VAR_GLOBAL
    (* OverrideMode *)
    {attribute 'pytmc' := 'pv: UED:RCC:VAC:OVRD_MODE'}
    xSystemOverrideMode_RCC	: BOOL := FALSE;

    (* Roughing Manifold Valvese *)

    {attribute 'pytmc' :=' pv: UED:RCC:VRC:01 '}
    {attribute 'TcLinkTo' := 	'.i_xClsLS	:=  TIID^Device 1 (EtherCAT)^Term 1 (EK1200)^RCC_E2 (EL1004)^Channel 1^Input;
                                .q_xOPN_DO	:=	TIID^Device 1 (EtherCAT)^Term 1 (EK1200)^RCC_E1 (EL2004)^Channel 1^Output'}
    RCC_VRC_01 : FB_VRC_NC_ClsLS;

    (* Roughing Manifold Valvese *)

    {attribute 'pytmc' :=' pv: UED:RCC:VRC:02 '}
    {attribute 'TcLinkTo' := 	'.i_xOpnLS	:= 	TIID^Device 1 (EtherCAT)^Term 1 (EK1200)^RCC_E2 (EL1004)^Channel 3^Input;
                                 .i_xClsLS	:=	TIID^Device 1 (EtherCAT)^Term 1 (EK1200)^RCC_E2 (EL1004)^Channel 4^Input;
                                .q_xOPN_DO	:=	TIID^Device 1 (EtherCAT)^Term 1 (EK1200)^RCC_E1 (EL2004)^Channel 2^Output'}
    RCC_VRC_02 : FB_VRC;

    (* Roughing Manifold Valvese *)

    {attribute 'pytmc' :=' pv: UED:RCC:VRC:03 '}
    {attribute 'TcLinkTo' := 	'.i_xClsLS	:=	TIID^Device 1 (EtherCAT)^Term 1 (EK1200)^RCC_E3 (EL1004)^Channel 1^Input;
                                .q_xOPN_DO	:= 	TIID^Device 1 (EtherCAT)^Term 1 (EK1200)^RCC_E1 (EL2004)^Channel 3^Output'}
    RCC_VRC_03 : FB_VRC_NC_ClsLS;

    (* Roughing Manifold Valvese *)

    {attribute 'pytmc' :=' pv: UED:RCC:VRC:04 '}
    {attribute 'TcLinkTo' := 	'.i_xClsLS	:=	TIID^Device 1 (EtherCAT)^Term 1 (EK1200)^RCC_E3 (EL1004)^Channel 1^Input;
                                .q_xOPN_DO	:=  TIID^Device 1 (EtherCAT)^Term 1 (EK1200)^RCC_E1 (EL2004)^Channel 4^Output'}
    RCC_VRC_04 : FB_VRC_NC_ClsLS;


    {attribute 'pytmc' :=' pv: UED:RCC:GCP:01 '}
    {attribute 'TcLinkTo' := 	'.xPress_OK		:=	TIID^Device 1 (EtherCAT)^Term 1 (EK1200)^Term 2 (EK1122)^Hoffman Box Vac EK1 (EK1100)^VLS_RCC (EK1122)^RCC_GPI (901P)^TXPDO Combined^Combination Gauge Reading Valid;
                                 .xOverrange	:=	TIID^Device 1 (EtherCAT)^Term 1 (EK1200)^Term 2 (EK1122)^Hoffman Box Vac EK1 (EK1100)^VLS_RCC (EK1122)^RCC_GPI (901P)^TXPDO Combined^Combination Gauge Overrange Exceeded;
                                .xUnderrange 	:= TIID^Device 1 (EtherCAT)^Term 1 (EK1200)^Term 2 (EK1122)^Hoffman Box Vac EK1 (EK1100)^VLS_RCC (EK1122)^RCC_GPI (901P)^TXPDO Combined^Combination Gauge Underrange Exceeded;
                                .i_iPRESS_R 	:= TIID^Device 1 (EtherCAT)^Term 1 (EK1200)^Term 2 (EK1122)^Hoffman Box Vac EK1 (EK1100)^VLS_RCC (EK1122)^RCC_GPI (901P)^TXPDO Combined^Combination Gauge Active Value;
                                .bWcstate 		:= TIID^Device 1 (EtherCAT)^Term 1 (EK1200)^Term 2 (EK1122)^Hoffman Box Vac EK1 (EK1100)^VLS_RCC (EK1122)^RCC_GPI (901P)^WcState^WcState' }
    RCC_GCP_01 : FB_901_ECAT;


    {attribute 'pytmc' :=' pv: UED:RCC:TC:01 '}
    {attribute 'TcLinkTo' := ' .bError 		:=	TIID^Device 1 (EtherCAT)^Term 1 (EK1200)^RCC_TC (EL3314)^TC Inputs Channel 1^Status^Error;
                               .bUnderrange :=	TIID^Device 1 (EtherCAT)^Term 1 (EK1200)^RCC_TC (EL3314)^TC Inputs Channel 1^Status^Underrange;
                               .bOverrange 	:=	TIID^Device 1 (EtherCAT)^Term 1 (EK1200)^RCC_TC (EL3314)^TC Inputs Channel 1^Status^Overrange ;
                               .iRaw		:= TIID^Device 1 (EtherCAT)^Term 1 (EK1200)^RCC_TC (EL3314)^TC Inputs Channel 1^Value '}
   RCC_STC_01 : FB_TempSensor;
END_VAR

(* stored: Version 1.1.0.1, ProductVersion 3.1.4024.12
   GVL GVL_RCC: Id {e34435c6-157b-4cae-9082-5ecee20695fb} *)
